SUBAPPLICATION Uebung_070d_AUI (* WBSD auf UT ausgeben mit AR_Timeout_Zero (Adapter Version) *)
  (* Standard: 61499-2; Description: Copyright (c) 2026 Meisterschulen am Ostbahnhof This program and the accompanying materials are made available under the terms of the Eclipse Public License 2.0 which is available at https://www.eclipse.org/legal/epl-2.0/ SPDX-License-Identifier: EPL-2.0 *)
  (* Version 1.0, 2026-09-17, Franz Höpfinger, Meisterschulen am Ostbahnhof, WBSD mit PHYS Skalierung und AR_Timeout_Zero Fendt-Schaltung (Adapter Version, analog Krauternter TECU_WBSD.SUB) *)
  PACKAGE Uebungen;
  IMPORT Uebungen::const::UT::TECU::DefaultPool_TECU_Numeric::NumberVariable_Wheel_based_machine_speed_N;
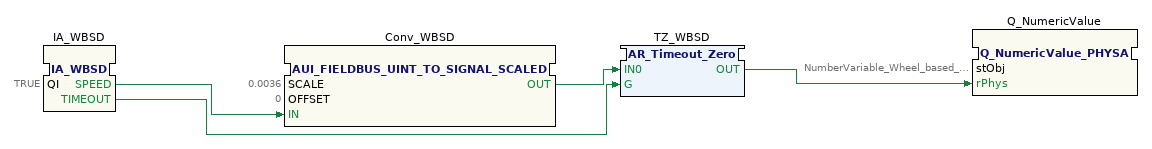
  FBS
    IA_WBSD : isobus::tecu::IA_WBSD(QI := TRUE);
    Conv_WBSD : logiBUS::signalprocessing::fieldbus::AUI_FIELDBUS_UINT_TO_SIGNAL_SCALED(SCALE := 0.0036, OFFSET := 0);
    Q_NumericValue : isobus::UT::Q::Q_NumericValue_PHYSA(stObj := NumberVariable_Wheel_based_machine_speed_N);
  END_FBS
  SUBAPPS
    TZ_WBSD : MyLib::sys::AR_Timeout_Zero;
  END_SUBAPPS
  ADAPTER_CONNECTIONS
    IA_WBSD.SPEED TO Conv_WBSD.IN;
    Conv_WBSD.OUT TO TZ_WBSD.IN0;
    IA_WBSD.TIMEOUT TO TZ_WBSD.G;
    TZ_WBSD.OUT TO Q_NumericValue.rPhys;
  END_CONNECTIONS
END_SUBAPPLICATION
